// TIA Portal V17 export
// export: Created 2024-09-02T12:50:30.1091245Z, ExportSetting WithDefaults, DisplayName Totally Integrated Automation Portal, DisplayVersion V17, DisplayName TIA Portal Openness, DisplayVersion V17, DisplayName TIA Portal Version Control Interface, DisplayVersion V17, DisplayName STEP 7 Professional, DisplayVersion V17, DisplayName STEP 7 Safety, DisplayVersion V17, DisplayName WinCC Professional, DisplayVersion V17
TYPE "typeSegmentanzeige"
TITLE = Segment display BNI IOL-802 / Segmentanzeige BNI IOL-802
// stored: IsFailsafeCompliant false
   STRUCT
      Farbe_GN_S1 { ExternalWritable := 'False'} : Bool;   // Segment Farbe / Segment Color
      Farbe_RD_S1 { ExternalWritable := 'False'} : Bool;   // Segment Farbe / Segment Color
      Farbe_BU_S1 { ExternalWritable := 'False'} : Bool;   // Segment Farbe / Segment Color
      Blinken_S1 { ExternalWritable := 'False'} : Bool;   // Segment Blinken ein / Segment Flashing on
      Farbe_GN_S2 { ExternalWritable := 'False'} : Bool;   // Segment Farbe / Segment Color
      Farbe_RD_S2 { ExternalWritable := 'False'} : Bool;   // Segment Farbe / Segment Color
      Farbe_BU_S2 { ExternalWritable := 'False'} : Bool;   // Segment Farbe / Segment Color
      Blinken_S2 { ExternalWritable := 'False'} : Bool;   // Segment Blinken ein / Segment Flashing on
      Farbe_GN_S3 { ExternalWritable := 'False'} : Bool;   // Segment Farbe / Segment Color
      Farbe_RD_S3 { ExternalWritable := 'False'} : Bool;   // Segment Farbe / Segment Color
      Farbe_BU_S3 { ExternalWritable := 'False'} : Bool;   // Segment Farbe / Segment Color
      Blinken_S3 { ExternalWritable := 'False'} : Bool;   // Segment Blinken ein / Segment Flashing on
      Farbe_GN_S4 { ExternalWritable := 'False'} : Bool;   // Segment Farbe / Segment Color
      Farbe_RD_S4 { ExternalWritable := 'False'} : Bool;   // Segment Farbe / Segment Color
      Farbe_BU_S4 { ExternalWritable := 'False'} : Bool;   // Segment Farbe / Segment Color
      Blinken_S4 { ExternalWritable := 'False'} : Bool;   // Segment Blinken ein / Segment Flashing on
      Farbe_GN_S5 { ExternalWritable := 'False'} : Bool;   // Segment Farbe / Segment Color
      Farbe_RD_S5 { ExternalWritable := 'False'} : Bool;   // Segment Farbe / Segment Color
      Farbe_BU_S5 { ExternalWritable := 'False'} : Bool;   // Segment Farbe / Segment Color
      Blinken_S5 { ExternalWritable := 'False'} : Bool;   // Segment Blinken ein / Segment Flashing on
      Reserve { ExternalWritable := 'False'} : Bool;
      Sync_Start { ExternalWritable := 'False'} : Bool;   // Zeitsynchronisierung starten / Start time synchronization
      Sync_Impuls { ExternalWritable := 'False'} : Bool;   // Zeitsynchronisierung impuls / Time synchronization pulse
      Summer_ein { ExternalWritable := 'False'} : Bool;   // Summer ein / Buzzer on
   END_STRUCT;
END_TYPE
